Yaskawa INFORM job: R2_BATVER2(-70,-90)AWOK.JBI

/JOB
//NAME R2_BATVER2(-70,-90)AWOK
///FOLDERNAME AWOK
//POS
///NPOS 163,163,0,5,0,0
///TOOL 0
///POSTYPE PULSE
///PULSE
C00000=61039,912,-47721,-12007,108779,37931
C00001=66285,32079,14392,-14564,112438,636
C00002=65621,33252,19577,-14432,109811,720
C00003=65356,33831,21768,-14387,108744,754
C00004=62507,41993,30149,-14933,107297,-122
C00005=62339,41731,30964,-14912,106650,-101
C00006=62507,41993,30149,-14933,107297,-122
C00007=65356,33831,21768,-14387,108744,754
C00008=64979,23936,16054,-14327,107157,810
C00009=64288,25680,17729,-14472,106903,586
C00010=64979,23936,16054,-14327,107157,810
C00011=65356,33831,21768,-14387,108744,754
C00012=76650,65179,59604,-11127,103520,5448
C00013=76933,67396,62555,-11020,102893,5607
C00014=76650,65179,59604,-11127,103520,5448
C00015=62507,41993,30149,-14933,107297,-122
C00016=62759,41305,27816,-14982,108390,-169
C00017=63393,39887,22323,-15124,111072,-283
C00018=118318,52612,40654,25271,81461,-73295
C00019=119564,52009,43489,25259,79214,-73309
C00020=120067,51865,44737,25265,78296,-73318
C00021=121803,51866,44761,25067,77755,-72776
C00022=121801,51522,45410,25115,77231,-72890
C00023=121803,51866,44761,25067,77755,-72776
C00024=120067,51865,44737,25265,78296,-73318
C00025=120042,48941,44190,25364,77245,-73556
C00026=120767,48924,44180,25284,77020,-73329
C00027=120042,48941,44190,25364,77245,-73556
C00028=120067,51865,44737,25265,78296,-73318
C00029=120407,63172,60728,25606,74534,-74015
C00030=120409,65179,63338,25670,74013,-74131
C00031=120407,63172,60728,25606,74534,-74015
C00032=121803,51866,44761,25067,77755,-72776
C00033=121296,51967,43466,25061,78681,-72769
C00034=120039,52468,40517,25074,80947,-72759
C00035=119825,49521,37362,-10695,82981,-53362
C00036=120209,50578,42665,-10795,80357,-53002
C00037=120362,51138,44950,-10843,79279,-52854
C00038=120356,50803,45649,-10861,78686,-52804
C00039=120362,51138,44950,-10843,79279,-52854
C00040=120443,55493,50145,-10882,78347,-52744
C00041=120445,58011,53363,-10907,77673,-52683
C00042=120443,55493,50145,-10882,78347,-52744
C00043=121152,53531,48086,-10945,78697,-52526
C00044=121834,53551,48117,-11013,78781,-52295
C00045=121152,53531,48086,-10945,78697,-52526
C00046=120999,52905,45716,-10894,79793,-52677
C00047=120618,51703,40233,-10788,82452,-53042
C00048=120473,51534,40147,-7135,83632,-50679
C00049=119092,49853,38858,26811,94834,-28763
C00050=117654,48102,37515,62184,106506,-5927
C00051=119888,49337,40582,62056,104469,-6071
C00052=120779,49927,41918,62014,103647,-6135
C00053=121515,49934,41936,62090,103175,-6011
C00054=120779,49927,41918,62014,103647,-6135
C00055=120412,51498,46747,61432,102809,-7103
C00056=120409,51785,47904,61255,102436,-7415
C00057=120412,51498,46747,61432,102809,-7103
C00058=120762,58431,54400,61213,102014,-7518
C00059=120764,60593,56840,61126,101816,-7679
C00060=120762,58431,54400,61213,102014,-7518
C00061=119893,57680,52847,61223,102849,-7434
C00062=117711,56087,49304,61270,104910,-7252
C00063=120729,53664,48209,60362,90886,40106
C00064=120731,53592,48129,60363,90890,40112
C00065=120732,53596,48133,60363,90890,40112
C00066=120906,53477,47753,60379,90870,40212
C00067=120737,52909,46098,60405,91349,40471
C00068=120316,53039,46469,60380,91530,40333
C00069=120884,53531,47939,60374,90840,40172
C00070=120732,53591,48128,60363,90890,40112
C00071=120732,53586,48122,60363,90891,40112
C00072=84698,56378,85785,35171,72174,-75436
C00073=84690,56271,85659,35166,72195,-75431
C00074=83027,27792,55307,40681,65778,-76398
C00075=82474,11517,44434,46729,56338,-78645
C00076=84160,53951,81707,34885,73419,-75237
C00077=84146,57749,87025,35100,72332,-75598
C00078=40685,4959,62266,27528,50532,-65290
C00079=46466,7401,61238,15330,52718,-61076
C00080=53708,-18565,35051,6276,42548,-57002
C00081=80566,27946,54769,40733,74240,-71241
C00082=120729,53658,48202,60362,90886,40107
C00083=120732,53586,48122,60363,90891,40112
C00084=120732,53590,48127,60363,90890,40112
C00085=121216,48798,43447,60402,90803,40364
C00086=120738,52903,46092,60405,91349,40471
C00087=120316,53033,46463,60380,91530,40333
C00088=120649,53283,47150,60377,91168,40274
C00089=120732,53586,48122,60363,90890,40112
C00090=120732,53580,48116,60363,90891,40113
C00091=93969,36532,52577,25566,110714,-40613
C00092=93964,36463,52505,25565,110724,-40613
C00093=93966,36477,52520,25566,110721,-40612
C00094=103842,25290,34157,14854,106745,-51915
C00095=93160,35996,51791,25225,111144,-40832
C00096=93519,35961,50866,25500,111538,-40597
C00097=103469,31990,41502,14628,105768,-52173
C00098=103089,39700,50220,14380,104475,-52468
C00099=102869,44686,56008,14229,103543,-52658
C00100=106797,22832,27569,6005,92316,-51957
C00101=106797,19989,18390,6055,96481,-51756
C00102=106797,19989,18390,6055,96481,-51756
C00103=120729,53662,48206,60973,81818,38390
C00104=120731,53590,48126,60971,81822,38396
C00105=120732,53594,48131,60971,81821,38395
C00106=120969,60466,55665,61086,81114,37990
C00107=120316,53037,46467,60907,82457,38620
C00108=120737,52907,46096,60882,82274,38758
C00109=117589,28291,29150,70668,90469,44270
C00110=114333,59672,68744,70035,96825,37495
C00111=114333,52714,52183,71172,99196,40406
C00112=114333,52714,52183,71172,99196,40406
C00113=120728,53745,48299,46872,97791,18406
C00114=120730,53673,48219,46873,97798,18411
C00115=120731,53674,48220,46873,97798,18411
C00116=120734,53609,47881,46895,97920,18472
C00117=120315,53114,46553,46923,98530,18561
C00118=120285,52139,47084,46808,97969,18274
C00119=120887,53567,47749,46054,98545,16857
C00120=120769,53596,48071,46013,98475,16768
C00121=119850,50104,44177,44548,94405,14514
C00122=119598,50013,44298,44518,94443,14412
C00123=117506,64097,65544,51116,97497,31231
C00124=112206,39413,48969,62120,100342,30156
C00125=111977,36482,45910,62148,100671,30274
C00126=115316,74650,90921,54864,108117,23431
C00127=112985,47782,61652,55421,111917,24650
C00128=112410,49443,55748,57098,114743,26510
C00129=120730,59879,52706,36408,68728,80702
C00130=120727,53927,48502,11034,106151,-61050
C00131=120730,53855,48421,11036,106163,-61048
C00132=120730,53855,48421,11036,106163,-61048
C00133=120730,53855,48421,11036,106163,-61048
C00134=120289,52533,46025,10966,107004,-61130
C00135=120874,56468,51135,11055,105822,-61027
C00136=120731,53815,48377,11036,106170,-61047
C00137=120731,53815,48377,11036,106170,-61047
C00138=120730,53815,48377,11036,106170,-61047
C00139=120731,51016,35282,-13941,85804,28522
C00140=120731,53534,48065,-21356,81011,21853
C00141=120732,53504,48031,-21356,81016,21852
C00142=120606,54302,48921,-21354,80856,21836
C00143=120950,52819,46056,-21331,81879,21778
C00144=121191,51326,45286,-21359,81668,21904
C00145=118879,69469,64198,-20764,88185,23557
C00146=121741,65875,61613,-20601,88664,24504
C00147=124845,68900,68891,-20623,95110,37615
C00148=134104,62401,67439,-18373,95240,41299
C00149=134104,58702,58571,-18552,98622,40782
C00150=135481,28796,11878,-19648,111614,39171
C00151=120727,62962,74819,-50624,75943,-2344
C00152=120727,62962,74819,-50624,75943,-64574
C00153=120729,62869,74710,-50621,75957,-64581
C00154=120730,62829,74662,-50619,75963,-64584
C00155=121502,26811,41007,-59205,62079,-58889
C00156=121182,64773,76463,-50603,76136,-64446
C00157=120987,61333,71630,-50414,76816,-64923
C00158=125744,21235,37921,-59733,64144,-57644
C00159=129553,74176,99619,-64295,61162,-52125
C00160=140879,17588,39239,-49360,57823,-60962
C00161=140879,9127,19117,-46085,63345,-64036
C00162=140879,1661,-16971,-41683,37099,-70140
BC00000=79328,124639,709625
BC00001=25113,42642,621063
BC00002=25113,42642,621063
BC00003=25113,42642,621063
BC00004=25113,42642,621063
BC00005=25113,42642,621063
BC00006=25113,42642,621063
BC00007=25113,42642,621063
BC00008=25113,42642,621063
BC00009=25113,42642,621063
BC00010=25113,42642,621063
BC00011=25113,42642,621063
BC00012=25113,42642,621063
BC00013=25113,42642,621063
BC00014=25113,42642,621063
BC00015=25113,42642,621063
BC00016=25113,42642,621063
BC00017=25113,42642,621063
BC00018=110747,234165,735656
BC00019=110747,234165,735656
BC00020=110747,234165,735656
BC00021=110747,234165,735656
BC00022=110747,234165,735656
BC00023=110747,234165,735656
BC00024=110747,234165,735656
BC00025=110747,234165,735656
BC00026=110747,234165,735656
BC00027=110747,234165,735656
BC00028=110747,234165,735656
BC00029=110747,234165,735656
BC00030=110747,234165,735656
BC00031=110747,234165,735656
BC00032=110747,234165,735656
BC00033=110747,234165,735656
BC00034=110747,234165,735656
BC00035=123779,146523,599461
BC00036=123779,146523,599461
BC00037=123779,146523,599461
BC00038=123779,146523,599461
BC00039=123779,146523,599461
BC00040=123779,146523,599461
BC00041=123779,146523,599461
BC00042=123779,146523,599461
BC00043=123779,146523,599461
BC00044=123779,146523,599461
BC00045=123779,146523,599461
BC00046=123779,146523,599461
BC00047=123779,146523,599461
BC00048=125038,140133,670722
BC00049=136728,80777,684478
BC00050=148910,18928,613463
BC00051=148910,18928,613463
BC00052=148910,18928,613463
BC00053=148910,18928,613463
BC00054=148910,18928,613463
BC00055=148910,18928,613463
BC00056=148910,18928,613463
BC00057=148910,18928,613463
BC00058=148910,18928,613463
BC00059=148910,18928,613463
BC00060=148910,18928,613463
BC00061=148910,18928,613463
BC00062=148910,18928,613463
BC00063=147878,97034,778223
BC00064=148299,97037,670698
BC00065=143506,97519,649294
BC00066=142080,97663,642923
BC00067=141589,97712,640732
BC00068=141589,97712,640732
BC00069=141851,163534,632925
BC00070=143768,163341,641487
BC00071=148561,162859,662891
BC00072=30249,0,1048172
BC00073=30671,0,940646
BC00074=27406,0,930849
BC00075=24732,0,922821
BC00076=22356,0,915693
BC00077=22356,0,915693
BC00078=24732,0,922821
BC00079=24732,1,922818
BC00080=24732,1,922818
BC00081=110050,92187,729884
BC00082=148122,158442,770940
BC00083=148544,158446,663414
BC00084=143751,158927,642010
BC00085=143152,158987,639333
BC00086=141834,159120,633449
BC00087=141834,159120,633449
BC00088=142096,224942,625642
BC00089=144013,224749,634203
BC00090=148806,224267,655607
BC00091=72055,165764,887383
BC00092=72476,165768,779858
BC00093=65883,167506,766061
BC00094=67508,167075,770959
BC00095=63246,168201,760542
BC00096=63246,168201,760542
BC00097=86557,135743,728984
BC00098=107130,101903,683650
BC00099=119568,81443,656241
BC00100=119568,81443,656239
BC00101=119568,81443,656239
BC00102=119568,81443,656239
BC00103=147935,121435,775167
BC00104=148356,121439,667642
BC00105=143558,120583,646395
BC00106=142543,120402,641902
BC00107=141639,120240,637897
BC00108=141639,120240,637897
BC00109=142543,11865,641897
BC00110=142543,11699,641897
BC00111=142543,11699,641897
BC00112=142543,11699,641897
BC00113=133499,217689,819497
BC00114=133920,217692,711972
BC00115=129774,216994,689149
BC00116=128116,216715,680021
BC00117=128116,216715,680021
BC00118=128116,216715,680021
BC00119=133059,206606,669522
BC00120=133059,206606,669522
BC00121=133059,206606,669522
BC00122=133059,206606,669522
BC00123=133059,206606,669522
BC00124=132873,208284,669777
BC00125=132873,208284,669777
BC00126=132873,208284,669777
BC00127=132873,187050,669777
BC00128=132862,187215,669812
BC00129=131229,279477,711594
BC00130=91042,204091,852535
BC00131=91463,204094,745010
BC00132=88172,208453,725866
BC00133=86855,210197,718208
BC00134=86855,210197,718208
BC00135=86855,210197,718208
BC00136=94396,207836,700767
BC00137=95713,206093,708425
BC00138=99005,201734,727569
BC00139=161054,197537,684508
BC00140=165338,185769,680618
BC00141=169930,183167,660631
BC00142=171052,182533,655735
BC00143=171767,182127,652636
BC00144=171767,182127,652636
BC00145=139904,152139,613102
BC00146=139904,152139,613102
BC00147=139904,152139,613102
BC00148=139904,111233,613102
BC00149=139904,111233,613102
BC00150=139904,111233,613102
BC00151=127845,123910,803748
BC00152=127845,123910,803748
BC00153=127887,123915,696213
BC00154=132560,126066,675788
BC00155=134430,126926,667619
BC00156=134430,126926,667619
BC00157=134430,126926,667619
BC00158=134430,126926,667619
BC00159=134430,126926,667619
BC00160=134430,126926,667619
BC00161=134430,126926,667619
BC00162=134430,126926,667619
///POSTYPE BASE
///RECTAN
///RCONF 0,0,0,0,0,0,0,0,0,0,0,0,0,0,0,0,0,0,0,0,0,0,0,0
P00006=0.222,-3.123,-1.508,0.0000,0.0000,0.0000
P00021=-0.225,-6.128,-0.405,0.0000,0.0000,0.0000
P00022=0.222,-3.123,-1.508,0.0000,0.0000,0.0000
P00023=0.143,-0.036,0.682,0.0000,0.0000,0.0000
P00024=0.145,-0.552,1.326,0.0000,0.0000,0.0000
//INST
///DATE 2023/11/15 16:43
///ATTR SC,RW
///GROUP1 RB1,BS1
NOP
'SEARCHE DO POPRAWY R1 I R2
'SEARCHE DO POPRAWY R1 I R2
'SEARCHE DO POPRAWY R1 I R2
'SEARCHE DO POPRAWY R1 I R2
'TYLKO SPOINY W DOBRYCH MIEJSCACH
'R2_BATver2(-70,-90)1
'Path S1158
SFTOF
MOVJ C00000 BC00000 VJ=10.00
MOVJ C00001 BC00001 VJ=10.00
MOVJ C00002 BC00002 VJ=10.00
MOVL C00003 BC00003 V=100.0
MOVL C00004 BC00004 V=60.0
REFP 3 C00005 BC00005
CALL JOB:SEARCH-R1
SET P021 P006
SFTON P021
MOVL C00006 BC00006 V=60.0
MOVL C00007 BC00007 V=100.0
MOVL C00008 BC00008 V=60.0
REFP 3 C00009 BC00009
CALL JOB:SEARCH-R1
SET P021 P006
SFTON P021
MOVL C00010 BC00010 V=60.0
MOVL C00011 BC00011 V=100.0
MOVL C00012 BC00012 V=60.0
REFP 3 C00013 BC00013
CALL JOB:SEARCH-R1
SET P021 P006
SFTON P021
MOVL C00014 BC00014 V=60.0
MOVL C00015 BC00015 V=100.0
MOVL C00016 BC00016 V=100.0
MOVL C00017 BC00017 V=100.0
'Path S1159
SFTOF
MOVJ C00018 BC00018 VJ=10.00
MOVJ C00019 BC00019 VJ=10.00
MOVL C00020 BC00020 V=100.0
MOVL C00021 BC00021 V=60.0
REFP 3 C00022 BC00022
CALL JOB:SEARCH-R1
SET P022 P006
SFTON P022
MOVL C00023 BC00023 V=60.0
MOVL C00024 BC00024 V=100.0
MOVL C00025 BC00025 V=60.0
REFP 3 C00026 BC00026
CALL JOB:SEARCH-R1
SET P022 P006
SFTON P022
MOVL C00027 BC00027 V=60.0
MOVL C00028 BC00028 V=100.0
MOVL C00029 BC00029 V=60.0
REFP 3 C00030 BC00030
CALL JOB:SEARCH-R1
SET P022 P006
SFTON P022
MOVL C00031 BC00031 V=60.0
MOVL C00032 BC00032 V=100.0
MOVL C00033 BC00033 V=100.0
MOVL C00034 BC00034 V=100.0
'Path S1160
SFTOF
MOVJ C00035 BC00035 VJ=10.00
MOVJ C00036 BC00036 VJ=10.00
MOVL C00037 BC00037 V=60.0
REFP 3 C00038 BC00038
CALL JOB:SEARCH-R1
SET P023 P006
SFTON P023
MOVL C00039 BC00039 V=60.0
MOVL C00040 BC00040 V=60.0
REFP 3 C00041 BC00041
CALL JOB:SEARCH-R1
SET P023 P006
SFTON P023
MOVL C00042 BC00042 V=60.0
MOVL C00043 BC00043 V=60.0
REFP 3 C00044 BC00044
CALL JOB:SEARCH-R1
SET P023 P006
SFTON P023
MOVL C00045 BC00045 V=60.0
MOVL C00046 BC00046 V=100.0
MOVL C00047 BC00047 V=100.0
'Path S1162
SFTOF
MOVJ C00048 BC00048 VJ=10.00
MOVJ C00049 BC00049 VJ=10.00
MOVJ C00050 BC00050 VJ=10.00
MOVJ C00051 BC00051 VJ=10.00
MOVL C00052 BC00052 V=60.0
REFP 3 C00053 BC00053
CALL JOB:SEARCH-R1
SET P024 P006
SFTON P024
MOVL C00054 BC00054 V=60.0
MOVL C00055 BC00055 V=60.0
REFP 3 C00056 BC00056
CALL JOB:SEARCH-R1
SET P024 P006
SFTON P024
MOVL C00057 BC00057 V=60.0
MOVL C00058 BC00058 V=60.0
REFP 3 C00059 BC00059
CALL JOB:SEARCH-R1
SET P024 P006
SFTON P024
MOVL C00060 BC00060 V=60.0
MOVL C00061 BC00061 V=100.0
MOVL C00062 BC00062 V=100.0
'Path W1163
SFTOF
SFTON P022
MOVJ C00063 BC00063 VJ=10.00
MOVJ C00064 BC00064 VJ=10.00
MOVJ C00065 BC00065 VJ=10.00
MOVL C00066 BC00066 V=100.0 PL=0
REFP 1 C00067 BC00067
REFP 2 C00068 BC00068
MACRO1 MJ#(0) ARGF9
ARCON
SFTON P024
MOVL C00069 BC00069 V=12.5
ARCOF
MOVL C00070 BC00070 V=100.0
MOVL C00071 BC00071 V=100.0
SFTOF
'Path W1164
SFTOF
SFTON P024
MOVJ C00072 BC00072 VJ=10.00
MOVJ C00073 BC00073 VJ=10.00
MOVJ C00074 BC00074 VJ=10.00
MOVL C00075 BC00075 V=100.0 PL=0
REFP 1 C00076 BC00076
REFP 2 C00077 BC00077
MACRO1 MJ#(0) ARGF10
ARCON
SFTON P023
MOVL C00078 BC00078 V=13.3
MOVL C00079 BC00079 V=13.3
ARCOF
MOVL C00080 BC00080 V=100.0
MOVL C00081 BC00081 V=100.0
SFTOF
'Path W1165
SFTOF
SFTON P022
MOVJ C00082 BC00082 VJ=10.00
MOVJ C00083 BC00083 VJ=10.00
MOVJ C00084 BC00084 VJ=10.00
MOVL C00085 BC00085 V=100.0 PL=0
REFP 1 C00086 BC00086
REFP 2 C00087 BC00087
MACRO1 MJ#(0) ARGF10
ARCON
MOVL C00088 BC00088 V=13.3
ARCOF
MOVL C00089 BC00089 V=100.0
MOVL C00090 BC00090 V=100.0
SFTOF
'Path W1166
SFTOF
SFTON P022
MOVJ C00091 BC00091 VJ=10.00
MOVJ C00092 BC00092 VJ=10.00
MOVJ C00093 BC00093 VJ=10.00
MOVL C00094 BC00094 V=100.0 PL=0
REFP 1 C00095 BC00095
REFP 2 C00096 BC00096
MACRO1 MJ#(0) ARGF10
ARCON
MOVL C00097 BC00097 V=14.2
MOVL C00098 BC00098 V=11.7
MOVL C00099 BC00099 V=14.2
COMM SFTON P023
MOVL C00100 BC00100 V=13.3
ARCOF
MOVL C00101 BC00101 V=100.0
MOVL C00102 BC00102 V=100.0
SFTOF
'Path W1167
SFTOF
SFTON P024
MOVJ C00103 BC00103 VJ=10.00
MOVJ C00104 BC00104 VJ=10.00
MOVJ C00105 BC00105 VJ=10.00
MOVL C00106 BC00106 V=100.0 PL=0
REFP 1 C00107 BC00107
REFP 2 C00108 BC00108
MACRO1 MJ#(0) ARGF10
ARCON
MOVL C00109 BC00109 V=14.2
MOVL C00110 BC00110 V=14.2
ARCOF
MOVL C00111 BC00111 V=100.0
MOVL C00112 BC00112 V=100.0
SFTOF
PAUSE
'Path W1168
SFTOF
SFTON P022
MOVJ C00113 BC00113 VJ=10.00
MOVJ C00114 BC00114 VJ=10.00
MOVJ C00115 BC00115 VJ=10.00
MOVL C00116 BC00116 V=100.0 PL=0
REFP 1 C00117 BC00117
REFP 2 C00118 BC00118
MACRO1 MJ#(0) ARGF10
ARCON
MOVL C00119 BC00119 V=10.0
MOVL C00120 BC00120 V=13.3
MOVL C00121 BC00121 V=13.3
MOVL C00122 BC00122 V=10.0
MOVL C00123 BC00123 V=10.8
MOVL C00124 BC00124 V=13.3
MOVL C00125 BC00125 V=10.0
MOVL C00126 BC00126 V=10.0
MOVL C00127 BC00127 V=14.2
ARCOF
MOVL C00128 BC00128 V=100.0
MOVL C00129 BC00129 V=100.0
'Path W1169
SFTOF
COMM SFTON P022
COMM MOVJ C00130 BC00130 VJ=100.00
COMM MOVJ C00131 BC00131 VJ=100.00
COMM MOVJ C00132 BC00132 VJ=100.00
COMM MOVL C00133 BC00133 V=100.0 PL=0
COMM REFP 1 C00134 BC00134
COMM REFP 2 C00135 BC00135
COMM MACRO1 MJ#(0) ARGF0
COMM ARCON
COMM MOVL C00136 BC00136 V=10.0
COMM ARCOF
COMM MOVL C00137 BC00137 V=400.0
COMM MOVL C00138 BC00138 V=1000.0
COMM SFTOF
'
'Path W1170
SFTOF
SFTON P021
MOVJ C00139 BC00139 VJ=10.00
MOVJ C00140 BC00140 VJ=10.00
MOVJ C00141 BC00141 VJ=10.00
MOVL C00142 BC00142 V=100.0 PL=0
REFP 1 C00143 BC00143
REFP 2 C00144 BC00144
MACRO1 MJ#(0) ARGF10
ARCON
MOVL C00145 BC00145 V=13.3
MOVL C00146 BC00146 V=13.3
MOVL C00147 BC00147 V=13.3
MOVL C00148 BC00148 V=13.3
ARCOF
MOVL C00149 BC00149 V=100.0
MOVL C00150 BC00150 V=100.0
MOVJ C00151 BC00151 VJ=10.00
SFTOF
'Path W1171
SFTON P021
MOVJ C00152 BC00152 VJ=10.00
MOVJ C00153 BC00153 VJ=10.00
MOVL C00154 BC00154 V=100.0
MOVL C00155 BC00155 V=100.0 PL=0
REFP 1 C00156 BC00156
REFP 2 C00157 BC00157
MACRO1 MJ#(0) ARGF10
ARCON
MOVL C00158 BC00158 V=13.3
MOVL C00159 BC00159 V=13.3
MOVL C00160 BC00160 V=13.3
ARCOF
MOVL C00161 BC00161 V=100.0
PAUSE
MOVJ C00162 BC00162 VJ=10.00
SFTOF
END
